// TwinCAT 3 PLC project APRProject2
// ProgramVersion: 3.1.4023.0
// libraries:
//   Tc2_Standard, * (Beckhoff Automation GmbH)
//   Tc2_System, * (Beckhoff Automation GmbH)
//   Tc3_Module, * (Beckhoff Automation GmbH)
// project tree:
//   DUTs/ sftDiModule.TcDUT (not stored), sftDoModule.TcDUT (not stored)
//   / GlobalTextList.TcGTLO, PlcTask.TcTTO, Visualization Manager.TcVMO (not stored), VISU_TASK.TcTTO
//   GVLs/ GVL.TcGVL (not stored), IO.TcGVL
//   POUs/ MAIN.TcPOU (not stored), sftDiCondAck.TcPOU (not stored), sftDiRunAck.TcPOU (not stored)
//   VISUs/ Visualization_1.TcVIS (not stored)
// real-time tasks:
//   TASK PlcTask: cycle T#10ms, priority 20, ADS port 350
//   TASK VISU_TASK: cycle T#200000us, priority 30, ADS port 351
// I/O:
//   DEVICE Device 1 (Beckhoff CCAT)
//   DEVICE Device 2 (EtherCAT), AmsNetId 5.52.95.234.3.1
//     Term 8 (EK1200) [EK1200-5000 EtherCAT Power supply (2A E-Bus)]
//       Term 2 (EL2008) [EL2008 8Ch. Dig. Output 24V, 0.5A]
//       Term 3 (EL2008) [EL2008 8Ch. Dig. Output 24V, 0.5A]
//       Term 4 (EL4021) [EL4021 1Ch. Ana. Output 4-20mA, 12bit]
//       Term 5 (EL4021) [EL4021 1Ch. Ana. Output 4-20mA, 12bit]
//       Term 6 (EL3021) [EL3021 1Ch. Ana. Input 4-20mA DIFF]
//       Term 7 (EL2008) [EL2008 8Ch. Dig. Output 24V, 0.5A]
//       Box 15 (BK1250)

CONFIGURATION APRProject2
    RESOURCE PLC ON TwinCAT3
        TASK PlcTask(INTERVAL := T#10ms, PRIORITY := 20);
        TASK VISU_TASK(INTERVAL := T#200000us, PRIORITY := 30);
        PROGRAM MAIN WITH PlcTask : MAIN;
        PROGRAM VisuElems_Visu_Prg WITH VISU_TASK : VisuElems.Visu_Prg;
    END_RESOURCE
END_CONFIGURATION

// ---- GVLs/IO.TcGVL
{attribute 'qualified_only'}
VAR_GLOBAL
	(* *) (* *) (* *) (* *) (* *) (* *) (* *) (* *) (* *) (* *) (* *) (* *) (* *)
	QualAck AT %I*:BOOL:=TRUE;
	(* *) (* *) (* *) (* *) (* *) (* *) (* *) (* *) (* *) (* *) (* *) (* *) (* *)
	p1_REF AT %I* : BOOL := FALSE; (*non-formal format: used with all dirxd*)
	p2_REF AT %I* : BOOL := FALSE; 
	p3_REF AT %I* : BOOL := FALSE;
	p4_REF AT %I* : BOOL := FALSE; 
	p5_REF AT %I* : BOOL := FALSE; 
	(* *) (* *) (* *) (* *) (* *) (* *) (* *) (* *) (* *) (* *) (* *) (* *) (* *)
	erikoismuuttujaSum AT %I* : BOOL := FALSE; 
	erikoismuuttujaDev AT %I* : BOOL := FALSE; 
	(* *) (* *) (* *) (* *) (* *) (* *) (* *) (* *) (* *) (* *) (* *) (* *) (* *)
	r1_REF AT %Q* : BOOL := FALSE; (*non-formal format: used with all dotxd*)
	r2_REF AT %Q* : BOOL := FALSE; 
	r3_REF AT %Q* : BOOL := FALSE;
	r4_REF AT %Q* : BOOL := FALSE; 
	r5_REF AT %Q* : BOOL := FALSE; (*non-formal format: used with all dotxd*)
	r6_REF AT %Q* : BOOL := FALSE; 
	(* *) (* *) (* *) (* *) (* *) (* *) (* *) (* *) (* *) (* *) (* *) (* *) (* *)
	fx1_REF AT %Q* : BOOL := FALSE; (* FMC 12 VDC BOOL 1|0 *) 
	fx2_REF AT %Q* : BOOL := FALSE; (* FMC 12 VDC BOOL 1|0 *) 
	fx3_REF AT %Q* : BOOL := FALSE; (* FMC 12 VDC BOOL 1|0 *) 
	fx4_REF AT %Q* : BOOL := FALSE; (* FMC 12 VDC BOOL 1|0 *) 
	fx5_REF AT %Q* : BOOL := FALSE; (* FMC 12 VDC BOOL 1|0 *) 	
	 (* *) (* *) (* *) (* *) (* *) (* *) (* *) (* *) (* *) (* *) (* *) (* *) (* *)
	v1_REF AT %Q* : BOOL := FALSE;
	v2_REF AT %Q* : BOOL := FALSE; 
	(* *) (* *) (* *) (* *) (* *) (* *) (* *) (* *) (* *) (* *) (* *) (* *) (* *)
	f1_REF AT %I*: INT; (* measured value (analog output for FMC, analog input for terminal, page 15) *) 
	f2_REF AT %I*: INT; (* measured value (analog output for FMC, analog input for terminal, page 15) *) 
	f3_REF AT %I*: INT; (* measured value (analog output for FMC, analog input for terminal, page 15) *) 
	f4_REF AT %I*: INT; (* measured value (analog output for FMC, analog input for terminal, page 15) *) 
	f5_REF AT %I*: INT; (* measured value (analog output for FMC, analog input for terminal, page 15) *) 
	(* *) (* *) (* *) (* *) (* *) (* *) (* *) (* *) (* *) (* *) (* *) (* *) (* *)
	k1_REF AT %Q*: INT :=7800; (* setpoint analog input for FMC, analog output for terminal, page 15) *)
	k2_REF AT %Q*: INT :=7800; (* setpoint analog input for FMC, analog output for terminal, page 15) *)
	k3_REF AT %Q*: INT :=7800; (* setpoint analog input for FMC, analog output for terminal, page 15) *)
	k4_REF AT %Q*: INT :=7800; (* setpoint analog input for FMC, analog output for terminal, page 15) *)
	k5_REF AT %Q*: INT :=7800; (* setpoint analog input for FMC, analog output for terminal, page 15) *)
	(* *) (* *) (* *) (* *) (* *) (* *) (* *) (* *) (* *) (* *) (* *) (* *) (* *)

	
	
	
	
	 // INT 15633 ja flow 30 ml/min 
	
	(* assign to term 3 KL3102 DATA IN *)

	
	

	


END_VAR

// ---- GlobalTextList.TcGTLO
TEXTLIST GlobalTextList
  493 = "'OPEN/CLOSE ALL VALVES'"
  538 = "'OPEN/CLOSE FC'"
  593 = "'OPEN/CLOSE FCs'"
  239 = "'OPEN/CLOSE VE1'"
  1 = "'OPEN/CLOSE VE4'"
  906 = "'OPEN/CLOSE VP1'"
  423 = "'OPEN/CLOSE VP2'"
  138 = "'OPEN/CLOSE VP3'"
  125 = "'OPEN/CLOSE VP4'"
  21 = "'OPEN/CLOSE VP5'"
  182 = "'OPEN/CLOSE VP6'"
  35 = "'Press to Control FC1'"
  833 = "'Press to Control Flow Controller 1'"
  317 = "'PRESS TO CTRL FC1'"
  163 = "'PRESS TO CTRL FC2'"
  485 = "'PRESS TO CTRL FC3'"
  294 = "'PRESS TO CTRL FC4'"
  835 = "'PRESS TO CTRL FC5'"
  487 = 'CLOSE ALL VALVES'
  463 = 'FIXED FLOW ML / MIN'
  723 = 'FIXED FLOW ML/MIN'
  318 = 'FLOW-COMMAND TOOL 2020'
  93 = 'ML/MIN'
  39 = 'OPEN ALL VALVES'
  225 = 'PRELIMINARY COMMAND TOOL '
  396 = 'preliminary command toolbox'
  826 = 'PRELIMINARY FLOW-COMMAND TOOL '
  526 = 'preliminary nuclear medicine command toolbox'
  181 = 'TEST ALL VALVES'
  216 = 'VE1'
  668 = 'VE4'
  925 = 'VP1'
  841 = 'VP2'
  95 = 'VP3'
  180 = 'VP4'
  719 = 'VP5'
  512 = 'VP6'
END_TEXTLIST
